LIN {X 0,Y 109.952,Z 432.134,A -85,B 0,C 180,E1 -30818.427,E2 -30818.427} C_VEL
LIN {X 0,Y 110.137,Z 438.588,A -85,B 0,C 180,E1 -30824.579,E2 -30824.579} C_VEL
LIN {X 0,Y 111.737,Z 444.355,A -85,B 0,C 180,E1 -30831.025,E2 -30831.025} C_VEL
LIN {X 0,Y 115.537,Z 449.975,A -85,B 0,C 180,E1 -30838.383,E2 -30838.383} C_VEL
LIN {X 0,Y 120.475,Z 454.059,A -85,B 0,C 180,E1 -30844.487,E2 -30844.487} C_VEL
LIN {X 0,Y 127.737,Z 457.673,A -85,B 0,C 180,E1 -30850.724,E2 -30850.724} C_VEL
LIN {X 0,Y 137.278,Z 460.508,A -85,B 0,C 180,E1 -30856.577,E2 -30856.577} C_VEL
LIN {X 0,Y 149.17,Z 462.456,A -85,B 0,C 180,E1 -30861.875,E2 -30861.875} C_VEL
LIN {X 0,Y 161.996,Z 463.408,A -85,B 0,C 180,E1 -30866.197,E2 -30866.197} C_VEL
LIN {X 0,Y 176.213,Z 463.483,A -85,B 0,C 180,E1 -30870,E2 -30870} C_VEL
LIN {X 0,Y 161.996,Z 463.408,A -85,B 0,C 180,E1 -30873.803,E2 -30873.803} C_VEL
LIN {X 0,Y 156.475,Z 463.174,A -85,B 0,C 180,E1 -30875.531,E2 -30875.531} C_VEL
LIN {X 0,Y 151.713,Z 462.95,A -85,B 0,C 180,E1 -30876.832,E2 -30876.832} C_VEL
LIN {X 0,Y 136.071,Z 462.302,A -85,B 0,C 180,E1 -30880.248,E2 -30880.248} C_VEL
LIN {X 0,Y 131.493,Z 461.883,A -85,B 0,C 180,E1 -30881.828,E2 -30881.828} C_VEL
LIN {X 0,Y 130.179,Z 461.635,A -85,B 0,C 180,E1 -30882.462,E2 -30882.462} C_VEL
LIN {X 0,Y 123.589,Z 460.079,A -85,B 0,C 180,E1 -30886.519,E2 -30886.519} C_VEL
LIN {X 0,Y 114.993,Z 456.749,A -85,B 0,C 180,E1 -30893.55,E2 -30893.55} C_VEL
LIN {X 0,Y 108.187,Z 451.587,A -85,B 0,C 180,E1 -30902.386,E2 -30902.386} C_VEL
LIN {X 0,Y 104.991,Z 446.653,A -85,B 0,C 180,E1 -30909.668,E2 -30909.668} C_VEL
LIN {X 0,Y 103.684,Z 440.506,A -85,B 0,C 180,E1 -30917.329,E2 -30917.329} C_VEL
LIN {X 0,Y 104.202,Z 433.989,A -85,B 0,C 180,E1 -30924.032,E2 -30924.032} C_VEL
LIN {X 0,Y 105.726,Z 427.305,A -85,B 0,C 180,E1 -30929.787,E2 -30929.787} C_VEL
LIN {X 0,Y 108.121,Z 419.38,A -85,B 0,C 180,E1 -30935.507,E2 -30935.507} C_VEL
LIN {X 0,Y 110.878,Z 411.533,A -85,B 0,C 180,E1 -30940.085,E2 -30940.085} C_VEL
LIN {X 0,Y 114.106,Z 402.226,A -85,B 0,C 180,E1 -30944.598,E2 -30944.598} C_VEL
LIN {X 0,Y 115.928,Z 396.712,A -85,B 0,C 180,E1 -30947.094,E2 -30947.094} C_VEL
LIN {X 0,Y 116.823,Z 392.5,A -85,B 0,C 180,E1 -30949.604,E2 -30949.604} C_VEL
LIN {X 0,Y 117.25,Z 390.258,A -85,B 0,C 180,E1 -30951.384,E2 -30951.384} C_VEL
LIN {X 0,Y 117.552,Z 388.558,A -85,B 0,C 180,E1 -30953.134,E2 -30953.134} C_VEL
LIN {X 0,Y 117.819,Z 386.305,A -85,B 0,C 180,E1 -30956.582,E2 -30956.582} C_VEL
LIN {X 0,Y 118.147,Z 384.922,A -85,B 0,C 180,E1 -30960.002,E2 -30960.002} C_VEL
LIN {X 0,Y 117.859,Z 385.79,A -85,B 0,C 180,E1 -30960.343,E2 -30960.343} C_VEL
LIN {X 0,Y 112.453,Z 398.556,A -85,B 0,C 180,E1 -30960.593,E2 -30960.593} C_VEL
LIN {X 0,Y 106.312,Z 409.458,A -85,B 0,C 180,E1 -30960.926,E2 -30960.926} C_VEL
LIN {X 0,Y 100.174,Z 418.396,A -85,B 0,C 180,E1 -30961.299,E2 -30961.299} C_VEL
LIN {X 0,Y 93.168,Z 426.918,A -85,B 0,C 180,E1 -30961.829,E2 -30961.829} C_VEL
LIN {X 0,Y 86.171,Z 434.13,A -85,B 0,C 180,E1 -30962.44,E2 -30962.44} C_VEL
LIN {X 0,Y 79.185,Z 440.325,A -85,B 0,C 180,E1 -30963.163,E2 -30963.163} C_VEL
LIN {X 0,Y 70.482,Z 446.858,A -85,B 0,C 180,E1 -30964.342,E2 -30964.342} C_VEL
LIN {X 0,Y 63.553,Z 451.36,A -85,B 0,C 180,E1 -30965.578,E2 -30965.578} C_VEL
LIN {X 0,Y 52.232,Z 457.31,A -85,B 0,C 180,E1 -30968.352,E2 -30968.352} C_VEL
LIN {X 0,Y 43.038,Z 461.18,A -85,B 0,C 180,E1 -30971.539,E2 -30971.539} C_VEL
LIN {X 0,Y 36.381,Z 463.552,A -85,B 0,C 180,E1 -30975.008,E2 -30975.008} C_VEL
LIN {X 0,Y 29.882,Z 465.355,A -85,B 0,C 180,E1 -30979.819,E2 -30979.819} C_VEL
LIN {X 0,Y 18.308,Z 467.822,A -85,B 0,C 180,E1 -30999.849,E2 -30999.849} C_VEL
LIN {X 0,Y 14.256,Z 468.423,A -85,B 0,C 180,E1 -31020.462,E2 -31020.462} C_VEL
LIN {X 0,Y 12.863,Z 468.588,A -85,B 0,C 180,E1 -31050,E2 -31050} C_VEL
LIN {X 0,Y 14.211,Z 468.422,A -85,B 0,C 180,E1 -31079.639,E2 -31079.639} C_VEL
LIN {X 0,Y 18.299,Z 467.822,A -85,B 0,C 180,E1 -31100.185,E2 -31100.185} C_VEL
LIN {X 0,Y 29.88,Z 465.354,A -85,B 0,C 180,E1 -31120.192,E2 -31120.192} C_VEL
LIN {X 0,Y 39.698,Z 462.4,A -85,B 0,C 180,E1 -31126.828,E2 -31126.828} C_VEL
LIN {X 0,Y 49.824,Z 458.409,A -85,B 0,C 180,E1 -31130.891,E2 -31130.891} C_VEL
LIN {X 0,Y 56.662,Z 455.192,A -85,B 0,C 180,E1 -31132.871,E2 -31132.871} C_VEL
LIN {X 0,Y 67.011,Z 449.168,A -85,B 0,C 180,E1 -31135.099,E2 -31135.099} C_VEL
LIN {X 0,Y 75.7,Z 443.075,A -85,B 0,C 180,E1 -31136.405,E2 -31136.405} C_VEL
LIN {X 0,Y 82.677,Z 437.38,A -85,B 0,C 180,E1 -31137.211,E2 -31137.211} C_VEL
LIN {X 0,Y 91.416,Z 428.834,A -85,B 0,C 180,E1 -31138.06,E2 -31138.06} C_VEL
LIN {X 0,Y 98.422,Z 420.664,A -85,B 0,C 180,E1 -31138.572,E2 -31138.572} C_VEL
LIN {X 0,Y 104.558,Z 412.16,A -85,B 0,C 180,E1 -31138.954,E2 -31138.954} C_VEL
LIN {X 0,Y 109.821,Z 403.451,A -85,B 0,C 180,E1 -31139.25,E2 -31139.25} C_VEL
LIN {X 0,Y 114.577,Z 393.86,A -85,B 0,C 180,E1 -31139.51,E2 -31139.51} C_VEL
LIN {X 0,Y 117.86,Z 385.789,A -85,B 0,C 180,E1 -31139.657,E2 -31139.657} C_VEL
LIN {X 0,Y 118.148,Z 384.921,A -85,B 0,C 180,E1 -31139.998,E2 -31139.998} C_VEL
LIN {X 0,Y 117.764,Z 386.797,A -85,B 0,C 180,E1 -31144.354,E2 -31144.354} C_VEL
LIN {X 0,Y 117.379,Z 389.446,A -85,B 0,C 180,E1 -31147.772,E2 -31147.772} C_VEL
LIN {X 0,Y 116.822,Z 392.502,A -85,B 0,C 180,E1 -31150.396,E2 -31150.396} C_VEL
LIN {X 0,Y 115.913,Z 396.746,A -85,B 0,C 180,E1 -31152.908,E2 -31152.908} C_VEL
LIN {X 0,Y 111.99,Z 408.401,A -85,B 0,C 180,E1 -31158.285,E2 -31158.285} C_VEL
LIN {X 0,Y 109.125,Z 416.544,A -85,B 0,C 180,E1 -31162.73,E2 -31162.73} C_VEL
LIN {X 0,Y 106.783,Z 423.698,A -85,B 0,C 180,E1 -31167.431,E2 -31167.431} C_VEL
LIN {X 0,Y 104.743,Z 431.236,A -85,B 0,C 180,E1 -31173.42,E2 -31173.42} C_VEL
LIN {X 0,Y 103.743,Z 438.536,A -85,B 0,C 180,E1 -31180.523,E2 -31180.523} C_VEL
LIN {X 0,Y 104.357,Z 444.73,A -85,B 0,C 180,E1 -31187.796,E2 -31187.796} C_VEL
LIN {X 0,Y 106.952,Z 450.021,A -85,B 0,C 180,E1 -31195.218,E2 -31195.218} C_VEL
LIN {X 0,Y 111.237,Z 454.336,A -85,B 0,C 180,E1 -31202.189,E2 -31202.189} C_VEL
LIN {X 0,Y 117.725,Z 457.962,A -85,B 0,C 180,E1 -31209.011,E2 -31209.011} C_VEL
LIN {X 0,Y 124.29,Z 460.275,A -85,B 0,C 180,E1 -31213.994,E2 -31213.994} C_VEL
LIN {X 0,Y 135.51,Z 462.499,A -85,B 0,C 180,E1 -31220.188,E2 -31220.188} C_VEL
LIN {X 0,Y 148.1,Z 463.65,A -85,B 0,C 180,E1 -31225.215,E2 -31225.215} C_VEL
LIN {X 0,Y 164.307,Z 463.8,A -85,B 0,C 180,E1 -31230,E2 -31230} C_VEL
LIN {X 0,Y 148.1,Z 463.65,A -85,B 0,C 180,E1 -31234.785,E2 -31234.785} C_VEL
LIN {X 0,Y 135.507,Z 462.502,A -85,B 0,C 180,E1 -31239.804,E2 -31239.804} C_VEL
LIN {X 0,Y 130.179,Z 461.635,A -85,B 0,C 180,E1 -31242.462,E2 -31242.462} C_VEL
LIN {X 0,Y 126.047,Z 461.085,A -85,B 0,C 180,E1 -31244.343,E2 -31244.343} C_VEL
LIN {X 0,Y 112.381,Z 459.488,A -85,B 0,C 180,E1 -31249.817,E2 -31249.817} C_VEL
LIN {X 0,Y 108.767,Z 458.593,A -85,B 0,C 180,E1 -31252.181,E2 -31252.181} C_VEL
LIN {X 0,Y 107.836,Z 458.22,A -85,B 0,C 180,E1 -31253.074,E2 -31253.074} C_VEL
LIN {X 0,Y 102.163,Z 454.476,A -85,B 0,C 180,E1 -31260.749,E2 -31260.749} C_VEL
LIN {X 0,Y 98.358,Z 449.147,A -85,B 0,C 180,E1 -31270.022,E2 -31270.022} C_VEL
LIN {X 0,Y 97.462,Z 442.32,A -85,B 0,C 180,E1 -31279.537,E2 -31279.537} C_VEL
LIN {X 0,Y 98.883,Z 435.097,A -85,B 0,C 180,E1 -31287.472,E2 -31287.472} C_VEL
LIN {X 0,Y 101.522,Z 427.548,A -85,B 0,C 180,E1 -31294.149,E2 -31294.149} C_VEL
LIN {X 0,Y 104.836,Z 419.614,A -85,B 0,C 180,E1 -31299.806,E2 -31299.806} C_VEL
LIN {X 0,Y 108.204,Z 411.945,A -85,B 0,C 180,E1 -31304.222,E2 -31304.222} C_VEL
LIN {X 0,Y 111.814,Z 403.367,A -85,B 0,C 180,E1 -31308.338,E2 -31308.338} C_VEL
LIN {X 0,Y 113.229,Z 399.587,A -85,B 0,C 180,E1 -31310.254,E2 -31310.254} C_VEL
LIN {X 0,Y 114.354,Z 395.938,A -85,B 0,C 180,E1 -31312.942,E2 -31312.942} C_VEL
LIN {X 0,Y 114.723,Z 394.314,A -85,B 0,C 180,E1 -31314.73,E2 -31314.73} C_VEL
LIN {X 0,Y 115.014,Z 393.125,A -85,B 0,C 180,E1 -31316.499,E2 -31316.499} C_VEL
LIN {X 0,Y 114.341,Z 394.573,A -85,B 0,C 180,E1 -31316.93,E2 -31316.93} C_VEL
LIN {X 0,Y 108.194,Z 406.499,A -85,B 0,C 180,E1 -31317.094,E2 -31317.094} C_VEL
LIN {X 0,Y 101.148,Z 417.069,A -85,B 0,C 180,E1 -31317.196,E2 -31317.196} C_VEL
LIN {X 0,Y 94.977,Z 424.806,A -85,B 0,C 180,E1 -31317.373,E2 -31317.373} C_VEL
LIN {X 0,Y 86.161,Z 433.937,A -85,B 0,C 180,E1 -31317.715,E2 -31317.715} C_VEL
LIN {X 0,Y 79.113,Z 440.132,A -85,B 0,C 180,E1 -31318.007,E2 -31318.007} C_VEL
LIN {X 0,Y 70.302,Z 446.665,A -85,B 0,C 180,E1 -31318.545,E2 -31318.545} C_VEL
LIN {X 0,Y 63.259,Z 451.166,A -85,B 0,C 180,E1 -31319.122,E2 -31319.122} C_VEL
LIN {X 0,Y 53.191,Z 456.446,A -85,B 0,C 180,E1 -31320.252,E2 -31320.252} C_VEL
LIN {X 0,Y 42.194,Z 460.986,A -85,B 0,C 180,E1 -31322.015,E2 -31322.015} C_VEL
LIN {X 0,Y 35.215,Z 463.358,A -85,B 0,C 180,E1 -31323.75,E2 -31323.75} C_VEL
LIN {X 0,Y 28.272,Z 465.161,A -85,B 0,C 180,E1 -31326.108,E2 -31326.108} C_VEL
LIN {X 0,Y 14.79,Z 467.629,A -85,B 0,C 180,E1 -31338.131,E2 -31338.131} C_VEL
LIN {X 0,Y 8.798,Z 468.23,A -85,B 0,C 180,E1 -31356.98,E2 -31356.98} C_VEL
LIN {X 0,Y 5.75,Z 468.395,A -85,B 0,C 180,E1 -31410,E2 -31410} C_VEL
LIN {X 0,Y 8.773,Z 468.229,A -85,B 0,C 180,E1 -31463.237,E2 -31463.237} C_VEL
LIN {X 0,Y 14.786,Z 467.628,A -85,B 0,C 180,E1 -31481.916,E2 -31481.916} C_VEL
LIN {X 0,Y 28.272,Z 465.161,A -85,B 0,C 180,E1 -31493.903,E2 -31493.903} C_VEL
LIN {X 0,Y 38.701,Z 462.206,A -85,B 0,C 180,E1 -31497.178,E2 -31497.178} C_VEL
LIN {X 0,Y 49.201,Z 458.215,A -85,B 0,C 180,E1 -31499.134,E2 -31499.134} C_VEL
LIN {X 0,Y 56.224,Z 454.998,A -85,B 0,C 180,E1 -31500.109,E2 -31500.109} C_VEL
LIN {X 0,Y 66.78,Z 448.975,A -85,B 0,C 180,E1 -31501.195,E2 -31501.195} C_VEL
LIN {X 0,Y 75.588,Z 442.882,A -85,B 0,C 180,E1 -31501.805,E2 -31501.805} C_VEL
LIN {X 0,Y 82.636,Z 437.188,A -85,B 0,C 180,E1 -31502.136,E2 -31502.136} C_VEL
LIN {X 0,Y 91.451,Z 428.641,A -85,B 0,C 180,E1 -31502.512,E2 -31502.512} C_VEL
LIN {X 0,Y 98.501,Z 420.471,A -85,B 0,C 180,E1 -31502.707,E2 -31502.707} C_VEL
LIN {X 0,Y 104.67,Z 411.967,A -85,B 0,C 180,E1 -31502.846,E2 -31502.846} C_VEL
LIN {X 0,Y 109.958,Z 403.259,A -85,B 0,C 180,E1 -31502.954,E2 -31502.954} C_VEL
LIN {X 0,Y 114.162,Z 394.978,A -85,B 0,C 180,E1 -31503.048,E2 -31503.048} C_VEL
LIN {X 0,Y 115.013,Z 393.127,A -85,B 0,C 180,E1 -31503.501,E2 -31503.501} C_VEL
LIN {X 0,Y 114.72,Z 394.322,A -85,B 0,C 180,E1 -31505.271,E2 -31505.271} C_VEL
LIN {X 0,Y 114.113,Z 396.913,A -85,B 0,C 180,E1 -31507.879,E2 -31507.879} C_VEL
LIN {X 0,Y 113.211,Z 399.616,A -85,B 0,C 180,E1 -31509.742,E2 -31509.742} C_VEL
LIN {X 0,Y 111.451,Z 404.34,A -85,B 0,C 180,E1 -31512.115,E2 -31512.115} C_VEL
LIN {X 0,Y 106.913,Z 415.068,A -85,B 0,C 180,E1 -31517.439,E2 -31517.439} C_VEL
LIN {X 0,Y 102.995,Z 423.979,A -85,B 0,C 180,E1 -31523.098,E2 -31523.098} C_VEL
LIN {X 0,Y 99.632,Z 432.65,A -85,B 0,C 180,E1 -31530.194,E2 -31530.194} C_VEL
LIN {X 0,Y 97.958,Z 438.802,A -85,B 0,C 180,E1 -31536.404,E2 -31536.404} C_VEL
LIN {X 0,Y 97.46,Z 444.88,A -85,B 0,C 180,E1 -31543.853,E2 -31543.853} C_VEL
LIN {X 0,Y 98.802,Z 450.027,A -85,B 0,C 180,E1 -31551.482,E2 -31551.482} C_VEL
LIN {X 0,Y 102.145,Z 454.481,A -85,B 0,C 180,E1 -31559.251,E2 -31559.251} C_VEL
LIN {X 0,Y 107.92,Z 458.249,A -85,B 0,C 180,E1 -31567,E2 -31567} C_VEL
LIN {X 0,Y 113.251,Z 460.373,A -85,B 0,C 180,E1 -31571.924,E2 -31571.924} C_VEL
LIN {X 0,Y 122.132,Z 462.491,A -85,B 0,C 180,E1 -31578.019,E2 -31578.019} C_VEL
LIN {X 0,Y 134.521,Z 463.877,A -85,B 0,C 180,E1 -31584.002,E2 -31584.002} C_VEL
LIN {X 0,Y 147.626,Z 464.245,A -85,B 0,C 180,E1 -31588.622,E2 -31588.622} C_VEL
LIN {X 0,Y 152.404,Z 464.117,A -85,B 0,C 180,E1 -31590,E2 -31590} C_VEL
LIN {X 0,Y 140.832,Z 464.131,A -85,B 0,C 180,E1 -31593.586,E2 -31593.586} C_VEL
LIN {X 0,Y 128.02,Z 463.258,A -85,B 0,C 180,E1 -31598.838,E2 -31598.838} C_VEL
LIN {X 0,Y 119.447,Z 461.928,A -85,B 0,C 180,E1 -31603.612,E2 -31603.612} C_VEL
LIN {X 0,Y 111.726,Z 459.855,A -85,B 0,C 180,E1 -31609.349,E2 -31609.349} C_VEL
LIN {X 0,Y 107.836,Z 458.22,A -85,B 0,C 180,E1 -31613.074,E2 -31613.074} C_VEL
LIN {X 0,Y 104.866,Z 457.195,A -85,B 0,C 180,E1 -31615.774,E2 -31615.774} C_VEL
LIN {X 0,Y 94.718,Z 454.51,A -85,B 0,C 180,E1 -31624.073,E2 -31624.073} C_VEL
LIN {X 0,Y 92.527,Z 453.084,A -85,B 0,C 180,E1 -31627.303,E2 -31627.303} C_VEL
LIN {X 0,Y 92.109,Z 452.483,A -85,B 0,C 180,E1 -31628.434,E2 -31628.434} C_VEL
LIN {X 0,Y 91.027,Z 448.147,A -85,B 0,C 180,E1 -31635.987,E2 -31635.987} C_VEL
LIN {X 0,Y 91.944,Z 441.68,A -85,B 0,C 180,E1 -31645.026,E2 -31645.026} C_VEL
LIN {X 0,Y 94.688,Z 434.482,A -85,B 0,C 180,E1 -31652.958,E2 -31652.958} C_VEL
LIN {X 0,Y 98.08,Z 427.57,A -85,B 0,C 180,E1 -31659.008,E2 -31659.008} C_VEL
LIN {X 0,Y 102.195,Z 419.847,A -85,B 0,C 180,E1 -31664.319,E2 -31664.319} C_VEL
LIN {X 0,Y 106.656,Z 411.289,A -85,B 0,C 180,E1 -31669.057,E2 -31669.057} C_VEL
LIN {X 0,Y 109.831,Z 404.885,A -85,B 0,C 180,E1 -31672.135,E2 -31672.135} C_VEL
LIN {X 0,Y 110.22,Z 403.943,A -85,B 0,C 180,E1 -31672.675,E2 -31672.675} C_VEL
LIN {X 0,Y 109.148,Z 405.657,A -85,B 0,C 180,E1 -31673.363,E2 -31673.363} C_VEL
LIN {X 0,Y 101.742,Z 416.876,A -85,B 0,C 180,E1 -31673.202,E2 -31673.202} C_VEL
LIN {X 0,Y 95.565,Z 424.614,A -85,B 0,C 180,E1 -31673.121,E2 -31673.121} C_VEL
LIN {X 0,Y 86.738,Z 433.743,A -85,B 0,C 180,E1 -31673.006,E2 -31673.006} C_VEL
LIN {X 0,Y 79.68,Z 439.938,A -85,B 0,C 180,E1 -31672.876,E2 -31672.876} C_VEL
LIN {X 0,Y 70.844,Z 446.471,A -85,B 0,C 180,E1 -31672.763,E2 -31672.763} C_VEL
LIN {X 0,Y 63.769,Z 450.972,A -85,B 0,C 180,E1 -31672.696,E2 -31672.696} C_VEL
LIN {X 0,Y 52.644,Z 456.689,A -85,B 0,C 180,E1 -31672.586,E2 -31672.586} C_VEL
LIN {X 0,Y 42.543,Z 460.793,A -85,B 0,C 180,E1 -31672.387,E2 -31672.387} C_VEL
LIN {X 0,Y 35.468,Z 463.165,A -85,B 0,C 180,E1 -31672.197,E2 -31672.197} C_VEL
LIN {X 0,Y 28.411,Z 464.968,A -85,B 0,C 180,E1 -31671.683,E2 -31671.683} C_VEL
LIN {X 0,Y 14.284,Z 467.435,A -85,B 0,C 180,E1 -31669.75,E2 -31669.75} C_VEL
LIN {X 0,Y 7.265,Z 468.037,A -85,B 0,C 180,E1 -31665.329,E2 -31665.329} C_VEL
LIN {X 0,Y 1.35,Z 468.202,A -85,B 0,C 180,E1 -31590,E2 -31590} C_VEL
LIN {X 0,Y 7.274,Z 468.036,A -85,B 0,C 180,E1 -31514.948,E2 -31514.948} C_VEL
LIN {X 0,Y 14.286,Z 467.434,A -85,B 0,C 180,E1 -31510.299,E2 -31510.299} C_VEL
LIN {X 0,Y 28.411,Z 464.968,A -85,B 0,C 180,E1 -31508.326,E2 -31508.326} C_VEL
LIN {X 0,Y 39.008,Z 462.012,A -85,B 0,C 180,E1 -31507.727,E2 -31507.727} C_VEL
LIN {X 0,Y 49.609,Z 458.021,A -85,B 0,C 180,E1 -31507.405,E2 -31507.405} C_VEL
LIN {X 0,Y 56.686,Z 454.805,A -85,B 0,C 180,E1 -31507.326,E2 -31507.326} C_VEL
LIN {X 0,Y 67.307,Z 448.782,A -85,B 0,C 180,E1 -31507.273,E2 -31507.273} C_VEL
LIN {X 0,Y 76.145,Z 442.689,A -85,B 0,C 180,E1 -31507.166,E2 -31507.166} C_VEL
LIN {X 0,Y 83.204,Z 436.995,A -85,B 0,C 180,E1 -31507.031,E2 -31507.031} C_VEL
LIN {X 0,Y 92.036,Z 428.448,A -85,B 0,C 180,E1 -31506.932,E2 -31506.932} C_VEL
LIN {X 0,Y 99.092,Z 420.278,A -85,B 0,C 180,E1 -31506.818,E2 -31506.818} C_VEL
LIN {X 0,Y 105.262,Z 411.774,A -85,B 0,C 180,E1 -31506.712,E2 -31506.712} C_VEL
LIN {X 0,Y 109.135,Z 405.681,A -85,B 0,C 180,E1 -31506.638,E2 -31506.638} C_VEL
LIN {X 0,Y 110.199,Z 403.982,A -85,B 0,C 180,E1 -31507.326,E2 -31507.326} C_VEL
LIN {X 0,Y 108.098,Z 408.486,A -85,B 0,C 180,E1 -31509.608,E2 -31509.608} C_VEL
LIN {X 0,Y 103.808,Z 416.836,A -85,B 0,C 180,E1 -31513.852,E2 -31513.852} C_VEL
LIN {X 0,Y 99.108,Z 425.627,A -85,B 0,C 180,E1 -31519.53,E2 -31519.53} C_VEL
LIN {X 0,Y 95.44,Z 432.915,A -85,B 0,C 180,E1 -31525.575,E2 -31525.575} C_VEL
LIN {X 0,Y 92.739,Z 439.22,A -85,B 0,C 180,E1 -31532.035,E2 -31532.035} C_VEL
LIN {X 0,Y 91.166,Z 445.137,A -85,B 0,C 180,E1 -31539.565,E2 -31539.565} C_VEL
LIN {X 0,Y 91.301,Z 450.221,A -85,B 0,C 180,E1 -31547.509,E2 -31547.509} C_VEL
LIN {X 0,Y 93.529,Z 454.579,A -85,B 0,C 180,E1 -31555.743,E2 -31555.743} C_VEL
LIN {X 0,Y 98.452,Z 458.531,A -85,B 0,C 180,E1 -31564.64,E2 -31564.64} C_VEL
LIN {X 0,Y 104.083,Z 460.927,A -85,B 0,C 180,E1 -31570.959,E2 -31570.959} C_VEL
LIN {X 0,Y 114.583,Z 463.243,A -85,B 0,C 180,E1 -31578.912,E2 -31578.912} C_VEL
LIN {X 0,Y 123.076,Z 464.184,A -85,B 0,C 180,E1 -31583.442,E2 -31583.442} C_VEL
LIN {X 0,Y 133.634,Z 464.587,A -85,B 0,C 180,E1 -31587.718,E2 -31587.718} C_VEL
LIN {X 0,Y 140.49,Z 464.434,A -85,B 0,C 180,E1 -31590,E2 -31590} C_VEL
LIN {X 0,Y 131.483,Z 464.526,A -85,B 0,C 180,E1 -31593.064,E2 -31593.064} C_VEL
LIN {X 0,Y 120.584,Z 464.003,A -85,B 0,C 180,E1 -31597.787,E2 -31597.787} C_VEL
LIN {X 0,Y 108.959,Z 462.222,A -85,B 0,C 180,E1 -31604.952,E2 -31604.952} C_VEL
LIN {X 0,Y 101.593,Z 460.006,A -85,B 0,C 180,E1 -31611.561,E2 -31611.561} C_VEL
LIN {X 0,Y 94.865,Z 455.993,A -85,B 0,C 180,E1 -31621.238,E2 -31621.238} C_VEL
LIN {X 0,Y 92.109,Z 452.483,A -85,B 0,C 180,E1 -31628.434,E2 -31628.434} C_VEL
LIN {X 0,Y 90.747,Z 450.813,A -85,B 0,C 180,E1 -31631.881,E2 -31631.881} C_VEL
LIN {X 0,Y 86.069,Z 446.561,A -85,B 0,C 180,E1 -31642.687,E2 -31642.687} C_VEL
LIN {X 0,Y 85.932,Z 444.588,A -85,B 0,C 180,E1 -31646.376,E2 -31646.376} C_VEL
LIN {X 0,Y 86.196,Z 443.807,A -85,B 0,C 180,E1 -31647.559,E2 -31647.559} C_VEL
LIN {X 0,Y 89.395,Z 437.538,A -85,B 0,C 180,E1 -31655.199,E2 -31655.199} C_VEL
LIN {X 0,Y 94.292,Z 429.466,A -85,B 0,C 180,E1 -31662.657,E2 -31662.657} C_VEL
LIN {X 0,Y 99.457,Z 421.341,A -85,B 0,C 180,E1 -31668.293,E2 -31668.293} C_VEL
LIN {X 0,Y 100.189,Z 420.084,A -85,B 0,C 180,E1 -31669.131,E2 -31669.131} C_VEL
LIN {X 0,Y 93.163,Z 428.255,A -85,B 0,C 180,E1 -31668.722,E2 -31668.722} C_VEL
LIN {X 0,Y 84.379,Z 436.801,A -85,B 0,C 180,E1 -31668.143,E2 -31668.143} C_VEL
LIN {X 0,Y 73.842,Z 445.123,A -85,B 0,C 180,E1 -31667.304,E2 -31667.304} C_VEL
LIN {X 0,Y 65.059,Z 450.779,A -85,B 0,C 180,E1 -31666.464,E2 -31666.464} C_VEL
LIN {X 0,Y 55.042,Z 456.046,A -85,B 0,C 180,E1 -31665.209,E2 -31665.209} C_VEL
LIN {X 0,Y 47.52,Z 459.36,A -85,B 0,C 180,E1 -31664.01,E2 -31664.01} C_VEL
LIN {X 0,Y 37.118,Z 462.971,A -85,B 0,C 180,E1 -31661.211,E2 -31661.211} C_VEL
LIN {X 0,Y 23.545,Z 466.17,A -85,B 0,C 180,E1 -31653.571,E2 -31653.571} C_VEL
LIN {X 0,Y 17.066,Z 467.241,A -85,B 0,C 180,E1 -31645.448,E2 -31645.448} C_VEL
LIN {X 0,Y 11.39,Z 467.843,A -85,B 0,C 180,E1 -31628.098,E2 -31628.098} C_VEL
LIN {X 0,Y 8.44,Z 468.01,A -85,B 0,C 180,E1 -31590,E2 -31590} C_VEL
LIN {X 0,Y 11.414,Z 467.843,A -85,B 0,C 180,E1 -31551.995,E2 -31551.995} C_VEL
LIN {X 0,Y 17.073,Z 467.241,A -85,B 0,C 180,E1 -31534.583,E2 -31534.583} C_VEL
LIN {X 0,Y 30.271,Z 464.775,A -85,B 0,C 180,E1 -31521.769,E2 -31521.769} C_VEL
LIN {X 0,Y 40.59,Z 461.818,A -85,B 0,C 180,E1 -31517.77,E2 -31517.77} C_VEL
LIN {X 0,Y 51.028,Z 457.827,A -85,B 0,C 180,E1 -31515.4,E2 -31515.4} C_VEL
LIN {X 0,Y 61.544,Z 452.695,A -85,B 0,C 180,E1 -31513.916,E2 -31513.916} C_VEL
LIN {X 0,Y 70.329,Z 447.433,A -85,B 0,C 180,E1 -31513.014,E2 -31513.014} C_VEL
LIN {X 0,Y 79.112,Z 441.12,A -85,B 0,C 180,E1 -31512.262,E2 -31512.262} C_VEL
LIN {X 0,Y 86.133,Z 435.175,A -85,B 0,C 180,E1 -31511.727,E2 -31511.727} C_VEL
LIN {X 0,Y 93.162,Z 428.255,A -85,B 0,C 180,E1 -31511.275,E2 -31511.275} C_VEL
LIN {X 0,Y 100.187,Z 420.084,A -85,B 0,C 180,E1 -31510.864,E2 -31510.864} C_VEL
LIN {X 0,Y 95.171,Z 428.026,A -85,B 0,C 180,E1 -31516.261,E2 -31516.261} C_VEL
LIN {X 0,Y 90.494,Z 435.565,A -85,B 0,C 180,E1 -31522.847,E2 -31522.847} C_VEL
LIN {X 0,Y 86.415,Z 443.315,A -85,B 0,C 180,E1 -31531.743,E2 -31531.743} C_VEL
LIN {X 0,Y 84.543,Z 449.726,A -85,B 0,C 180,E1 -31541.681,E2 -31541.681} C_VEL
LIN {X 0,Y 85.378,Z 454.613,A -85,B 0,C 180,E1 -31551.436,E2 -31551.436} C_VEL
LIN {X 0,Y 89.356,Z 458.807,A -85,B 0,C 180,E1 -31561.842,E2 -31561.842} C_VEL
LIN {X 0,Y 93.403,Z 460.947,A -85,B 0,C 180,E1 -31567.9,E2 -31567.9} C_VEL
LIN {X 0,Y 101.462,Z 463.165,A -85,B 0,C 180,E1 -31575.859,E2 -31575.859} C_VEL
LIN {X 0,Y 113.189,Z 464.541,A -85,B 0,C 180,E1 -31583.421,E2 -31583.421} C_VEL
LIN {X 0,Y 126.513,Z 464.807,A -85,B 0,C 180,E1 -31589.181,E2 -31589.181} C_VEL
LIN {X 0,Y 128.831,Z 464.745,A -85,B 0,C 180,E1 -31590,E2 -31590} C_VEL
LIN {X 0,Y 119.694,Z 464.822,A -85,B 0,C 180,E1 -31593.489,E2 -31593.489} C_VEL
LIN {X 0,Y 107.081,Z 463.973,A -85,B 0,C 180,E1 -31600.118,E2 -31600.118} C_VEL
LIN {X 0,Y 98.651,Z 462.513,A -85,B 0,C 180,E1 -31606.557,E2 -31606.557} C_VEL
LIN {X 0,Y 92.14,Z 460.392,A -85,B 0,C 180,E1 -31613.758,E2 -31613.758} C_VEL
LIN {X 0,Y 86.432,Z 456.265,A -85,B 0,C 180,E1 -31624.693,E2 -31624.693} C_VEL
LIN {X 0,Y 84.475,Z 451.478,A -85,B 0,C 180,E1 -31634.999,E2 -31634.999} C_VEL
LIN {X 0,Y 85.077,Z 446.713,A -85,B 0,C 180,E1 -31643.25,E2 -31643.25} C_VEL
LIN {X 0,Y 86.196,Z 443.807,A -85,B 0,C 180,E1 -31647.559,E2 -31647.559} C_VEL
LIN {X 0,Y 86.44,Z 442.413,A -85,B 0,C 180,E1 -31650.046,E2 -31650.046} C_VEL
LIN {X 0,Y 85.502,Z 439.043,A -85,B 0,C 180,E1 -31658.747,E2 -31658.747} C_VEL
LIN {X 0,Y 86.371,Z 437.319,A -85,B 0,C 180,E1 -31661.062,E2 -31661.062} C_VEL
LIN {X 0,Y 88.035,Z 434.965,A -85,B 0,C 180,E1 -31663.332,E2 -31663.332} C_VEL
LIN {X 0,Y 87.865,Z 434.982,A -85,B 0,C 180,E1 -31663.706,E2 -31663.706} C_VEL
LIN {X 0,Y 80.927,Z 440.927,A -85,B 0,C 180,E1 -31662.801,E2 -31662.801} C_VEL
LIN {X 0,Y 72.272,Z 447.24,A -85,B 0,C 180,E1 -31661.464,E2 -31661.464} C_VEL
LIN {X 0,Y 63.64,Z 452.501,A -85,B 0,C 180,E1 -31659.832,E2 -31659.832} C_VEL
LIN {X 0,Y 53.37,Z 457.633,A -85,B 0,C 180,E1 -31657.189,E2 -31657.189} C_VEL
LIN {X 0,Y 43.302,Z 461.624,A -85,B 0,C 180,E1 -31653.208,E2 -31653.208} C_VEL
LIN {X 0,Y 33.561,Z 464.582,A -85,B 0,C 180,E1 -31646.891,E2 -31646.891} C_VEL
LIN {X 0,Y 21.911,Z 467.047,A -85,B 0,C 180,E1 -31629.904,E2 -31629.904} C_VEL
LIN {X 0,Y 17.547,Z 467.65,A -85,B 0,C 180,E1 -31613.611,E2 -31613.611} C_VEL
LIN {X 0,Y 15.549,Z 467.817,A -85,B 0,C 180,E1 -31590,E2 -31590} C_VEL
LIN {X 0,Y 17.57,Z 467.65,A -85,B 0,C 180,E1 -31566.422,E2 -31566.422} C_VEL
LIN {X 0,Y 21.919,Z 467.047,A -85,B 0,C 180,E1 -31550.113,E2 -31550.113} C_VEL
LIN {X 0,Y 33.563,Z 464.582,A -85,B 0,C 180,E1 -31533.115,E2 -31533.115} C_VEL
LIN {X 0,Y 43.304,Z 461.624,A -85,B 0,C 180,E1 -31526.796,E2 -31526.796} C_VEL
LIN {X 0,Y 53.369,Z 457.633,A -85,B 0,C 180,E1 -31522.809,E2 -31522.809} C_VEL
LIN {X 0,Y 63.641,Z 452.501,A -85,B 0,C 180,E1 -31520.17,E2 -31520.17} C_VEL
LIN {X 0,Y 72.272,Z 447.24,A -85,B 0,C 180,E1 -31518.536,E2 -31518.536} C_VEL
LIN {X 0,Y 80.921,Z 440.927,A -85,B 0,C 180,E1 -31517.188,E2 -31517.188} C_VEL
LIN {X 0,Y 87.853,Z 434.983,A -85,B 0,C 180,E1 -31516.268,E2 -31516.268} C_VEL
LIN {X 0,Y 88.03,Z 434.966,A -85,B 0,C 180,E1 -31516.659,E2 -31516.659} C_VEL
LIN {X 0,Y 82.482,Z 442.715,A -85,B 0,C 180,E1 -31525.213,E2 -31525.213} C_VEL
LIN {X 0,Y 78.589,Z 449.926,A -85,B 0,C 180,E1 -31536.405,E2 -31536.405} C_VEL
LIN {X 0,Y 77.913,Z 454.583,A -85,B 0,C 180,E1 -31546.184,E2 -31546.184} C_VEL
LIN {X 0,Y 80.624,Z 459.081,A -85,B 0,C 180,E1 -31558.465,E2 -31558.465} C_VEL
LIN {X 0,Y 84.527,Z 461.44,A -85,B 0,C 180,E1 -31566.142,E2 -31566.142} C_VEL
LIN {X 0,Y 88.803,Z 462.864,A -85,B 0,C 180,E1 -31571.741,E2 -31571.741} C_VEL
LIN {X 0,Y 101.121,Z 464.785,A -85,B 0,C 180,E1 -31582.01,E2 -31582.01} C_VEL
LIN {X 0,Y 112.511,Z 465.186,A -85,B 0,C 180,E1 -31588.022,E2 -31588.022} C_VEL
LIN {X 0,Y 117.267,Z 465.056,A -85,B 0,C 180,E1 -31590,E2 -31590} C_VEL
LIN {X 0,Y 105.857,Z 465.007,A -85,B 0,C 180,E1 -31595.234,E2 -31595.234} C_VEL
LIN {X 0,Y 99.612,Z 464.684,A -85,B 0,C 180,E1 -31598.993,E2 -31598.993} C_VEL
LIN {X 0,Y 88.566,Z 462.8,A -85,B 0,C 180,E1 -31608.506,E2 -31608.506} C_VEL
LIN {X 0,Y 84.02,Z 461.224,A -85,B 0,C 180,E1 -31614.723,E2 -31614.723} C_VEL
LIN {X 0,Y 78.947,Z 457.333,A -85,B 0,C 180,E1 -31626.76,E2 -31626.76} C_VEL
LIN {X 0,Y 77.855,Z 453.539,A -85,B 0,C 180,E1 -31636.233,E2 -31636.233} C_VEL
LIN {X 0,Y 79.399,Z 448.009,A -85,B 0,C 180,E1 -31646.882,E2 -31646.882} C_VEL
LIN {X 0,Y 83.132,Z 441.707,A -85,B 0,C 180,E1 -31656.033,E2 -31656.033} C_VEL
LIN {X 0,Y 86.371,Z 437.319,A -85,B 0,C 180,E1 -31661.062,E2 -31661.062} C_VEL
LIN {X 0,Y 85.41,Z 438.095,A -85,B 0,C 180,E1 -31661.09,E2 -31661.09} C_VEL
LIN {X 0,Y 81.573,Z 441.77,A -85,B 0,C 180,E1 -31658.88,E2 -31658.88} C_VEL
LIN {X 0,Y 77.828,Z 445.591,A -85,B 0,C 180,E1 -31655.18,E2 -31655.18} C_VEL
LIN {X 0,Y 75.269,Z 448.303,A -85,B 0,C 180,E1 -31651.87,E2 -31651.87} C_VEL
LIN {X 0,Y 72.487,Z 451.757,A -85,B 0,C 180,E1 -31646.161,E2 -31646.161} C_VEL
LIN {X 0,Y 71.958,Z 452.745,A -85,B 0,C 180,E1 -31644.076,E2 -31644.076} C_VEL
LIN {X 0,Y 71.151,Z 456.799,A -85,B 0,C 180,E1 -31633.743,E2 -31633.743} C_VEL
LIN {X 0,Y 72.261,Z 459.353,A -85,B 0,C 180,E1 -31625.701,E2 -31625.701} C_VEL
LIN {X 0,Y 74.897,Z 461.5,A -85,B 0,C 180,E1 -31617.981,E2 -31617.981} C_VEL
LIN {X 0,Y 81.174,Z 463.741,A -85,B 0,C 180,E1 -31607.764,E2 -31607.764} C_VEL
LIN {X 0,Y 92.19,Z 465.166,A -85,B 0,C 180,E1 -31597.695,E2 -31597.695} C_VEL
LIN {X 0,Y 98.592,Z 465.473,A -85,B 0,C 180,E1 -31593.683,E2 -31593.683} C_VEL
LIN {X 0,Y 105.989,Z 465.362,A -85,B 0,C 180,E1 -31590,E2 -31590} C_VEL
LIN {X 0,Y 97.797,Z 465.439,A -85,B 0,C 180,E1 -31585.879,E2 -31585.879} C_VEL
LIN {X 0,Y 86.329,Z 464.603,A -85,B 0,C 180,E1 -31577.651,E2 -31577.651} C_VEL
LIN {X 0,Y 78.859,Z 463.079,A -85,B 0,C 180,E1 -31569.116,E2 -31569.116} C_VEL
LIN {X 0,Y 73.735,Z 460.696,A -85,B 0,C 180,E1 -31559.068,E2 -31559.068} C_VEL
LIN {X 0,Y 71.162,Z 456.799,A -85,B 0,C 180,E1 -31546.265,E2 -31546.265} C_VEL
LIN {X 0,Y 71.991,Z 452.703,A -85,B 0,C 180,E1 -31535.851,E2 -31535.851} C_VEL
LIN {X 0,Y 74.872,Z 448.093,A -85,B 0,C 180,E1 -31526.909,E2 -31526.909} C_VEL
LIN {X 0,Y 76.524,Z 445.892,A -85,B 0,C 180,E1 -31523.307,E2 -31523.307} C_VEL
LIN {X 0,Y 69.791,Z 450.391,A -85,B 0,C 180,E1 -31525.001,E2 -31525.001} C_VEL
LIN {X 0,Y 60.888,Z 455.367,A -85,B 0,C 180,E1 -31527.758,E2 -31527.758} C_VEL
LIN {X 0,Y 50.063,Z 460.214,A -85,B 0,C 180,E1 -31532.617,E2 -31532.617} C_VEL
LIN {X 0,Y 43.866,Z 462.583,A -85,B 0,C 180,E1 -31536.767,E2 -31536.767} C_VEL
LIN {X 0,Y 37.938,Z 464.388,A -85,B 0,C 180,E1 -31542.183,E2 -31542.183} C_VEL
LIN {X 0,Y 27.761,Z 466.854,A -85,B 0,C 180,E1 -31559.581,E2 -31559.581} C_VEL
LIN {X 0,Y 24.275,Z 467.456,A -85,B 0,C 180,E1 -31573.171,E2 -31573.171} C_VEL
LIN {X 0,Y 22.647,Z 467.624,A -85,B 0,C 180,E1 -31590,E2 -31590} C_VEL
LIN {X 0,Y 24.255,Z 467.457,A -85,B 0,C 180,E1 -31606.843,E2 -31606.843} C_VEL
LIN {X 0,Y 27.753,Z 466.854,A -85,B 0,C 180,E1 -31620.429,E2 -31620.429} C_VEL
LIN {X 0,Y 37.935,Z 464.388,A -85,B 0,C 180,E1 -31637.821,E2 -31637.821} C_VEL
LIN {X 0,Y 46.947,Z 461.431,A -85,B 0,C 180,E1 -31645.421,E2 -31645.421} C_VEL
LIN {X 0,Y 56.524,Z 457.439,A -85,B 0,C 180,E1 -31650.5,E2 -31650.5} C_VEL
LIN {X 0,Y 66.439,Z 452.307,A -85,B 0,C 180,E1 -31654.045,E2 -31654.045} C_VEL
LIN {X 0,Y 74.839,Z 447.046,A -85,B 0,C 180,E1 -31656.292,E2 -31656.292} C_VEL
LIN {X 0,Y 76.575,Z 445.888,A -85,B 0,C 180,E1 -31656.606,E2 -31656.606} C_VEL
LIN {X 0,Y 72.481,Z 451.702,A -85,B 0,C 180,E1 -31646.294,E2 -31646.294} C_VEL
LIN {X 0,Y 71.958,Z 452.745,A -85,B 0,C 180,E1 -31644.076,E2 -31644.076} C_VEL
LIN {X 0,Y 70.698,Z 454.879,A -85,B 0,C 180,E1 -31639.741,E2 -31639.741} C_VEL
LIN {X 0,Y 67.834,Z 458.333,A -85,B 0,C 180,E1 -31632.398,E2 -31632.398} C_VEL
LIN {X 0,Y 66.251,Z 461.115,A -85,B 0,C 180,E1 -31624.428,E2 -31624.428} C_VEL
LIN {X 0,Y 67.028,Z 462.248,A -85,B 0,C 180,E1 -31619.527,E2 -31619.527} C_VEL
LIN {X 0,Y 74.014,Z 464.529,A -85,B 0,C 180,E1 -31606.551,E2 -31606.551} C_VEL
LIN {X 0,Y 79.974,Z 465.366,A -85,B 0,C 180,E1 -31600.123,E2 -31600.123} C_VEL
LIN {X 0,Y 91.41,Z 465.759,A -85,B 0,C 180,E1 -31591.893,E2 -31591.893} C_VEL
LIN {X 0,Y 94.915,Z 465.662,A -85,B 0,C 180,E1 -31590,E2 -31590} C_VEL
LIN {X 0,Y 84.814,Z 465.631,A -85,B 0,C 180,E1 -31583.886,E2 -31583.886} C_VEL
LIN {X 0,Y 78.807,Z 465.287,A -85,B 0,C 180,E1 -31578.792,E2 -31578.792} C_VEL
LIN {X 0,Y 69.302,Z 463.308,A -85,B 0,C 180,E1 -31565.874,E2 -31565.874} C_VEL
LIN {X 0,Y 65.254,Z 460.777,A -85,B 0,C 180,E1 -31553.843,E2 -31553.843} C_VEL
LIN {X 0,Y 64.361,Z 458.555,A -85,B 0,C 180,E1 -31545.03,E2 -31545.03} C_VEL
LIN {X 0,Y 65.589,Z 454.96,A -85,B 0,C 180,E1 -31534.145,E2 -31534.145} C_VEL
LIN {X 0,Y 61.601,Z 456.625,A -85,B 0,C 180,E1 -31534.777,E2 -31534.777} C_VEL
LIN {X 0,Y 54.232,Z 460.02,A -85,B 0,C 180,E1 -31538.963,E2 -31538.963} C_VEL
LIN {X 0,Y 48.48,Z 462.389,A -85,B 0,C 180,E1 -31543.545,E2 -31543.545} C_VEL
LIN {X 0,Y 43.054,Z 464.194,A -85,B 0,C 180,E1 -31549.236,E2 -31549.236} C_VEL
LIN {X 0,Y 34.106,Z 466.66,A -85,B 0,C 180,E1 -31565.661,E2 -31565.661} C_VEL
LIN {X 0,Y 31.16,Z 467.263,A -85,B 0,C 180,E1 -31576.965,E2 -31576.965} C_VEL
LIN {X 0,Y 29.762,Z 467.431,A -85,B 0,C 180,E1 -31590,E2 -31590} C_VEL
LIN {X 0,Y 31.142,Z 467.263,A -85,B 0,C 180,E1 -31603.042,E2 -31603.042} C_VEL
LIN {X 0,Y 34.098,Z 466.66,A -85,B 0,C 180,E1 -31614.345,E2 -31614.345} C_VEL
LIN {X 0,Y 43.052,Z 464.194,A -85,B 0,C 180,E1 -31630.766,E2 -31630.766} C_VEL
LIN {X 0,Y 51.324,Z 461.237,A -85,B 0,C 180,E1 -31638.863,E2 -31638.863} C_VEL
LIN {X 0,Y 60.363,Z 457.245,A -85,B 0,C 180,E1 -31644.587,E2 -31644.587} C_VEL
LIN {X 0,Y 61.392,Z 456.736,A -85,B 0,C 180,E1 -31645.088,E2 -31645.088} C_VEL
LIN {X 0,Y 65.575,Z 454.966,A -85,B 0,C 180,E1 -31645.855,E2 -31645.855} C_VEL
LIN {X 0,Y 64.35,Z 458.554,A -85,B 0,C 180,E1 -31634.983,E2 -31634.983} C_VEL
LIN {X 0,Y 67.028,Z 462.248,A -85,B 0,C 180,E1 -31619.527,E2 -31619.527} C_VEL
LIN {X 0,Y 68.325,Z 463.31,A -85,B 0,C 180,E1 -31614.71,E2 -31614.71} C_VEL
LIN {X 0,Y 69.892,Z 464.809,A -85,B 0,C 180,E1 -31606.675,E2 -31606.675} C_VEL
LIN {X 0,Y 72.051,Z 465.651,A -85,B 0,C 180,E1 -31600.567,E2 -31600.567} C_VEL
LIN {X 0,Y 74.903,Z 465.946,A -85,B 0,C 180,E1 -31596.564,E2 -31596.564} C_VEL
LIN {X 0,Y 76.151,Z 466.015,A -85,B 0,C 180,E1 -31595.42,E2 -31595.42} C_VEL
LIN {X 0,Y 83.963,Z 465.96,A -85,B 0,C 180,E1 -31590,E2 -31590} C_VEL
LIN {X 0,Y 76.292,Z 466.025,A -85,B 0,C 180,E1 -31584.714,E2 -31584.714} C_VEL
LIN {X 0,Y 65.954,Z 465.137,A -85,B 0,C 180,E1 -31573.532,E2 -31573.532} C_VEL
LIN {X 0,Y 60.395,Z 463.628,A -85,B 0,C 180,E1 -31562.26,E2 -31562.26} C_VEL
LIN {X 0,Y 57.56,Z 460.827,A -85,B 0,C 180,E1 -31547.099,E2 -31547.099} C_VEL
LIN {X 0,Y 53.646,Z 462.195,A -85,B 0,C 180,E1 -31549.078,E2 -31549.078} C_VEL
LIN {X 0,Y 48.678,Z 464.001,A -85,B 0,C 180,E1 -31554.725,E2 -31554.725} C_VEL
LIN {X 0,Y 40.725,Z 466.466,A -85,B 0,C 180,E1 -31569.81,E2 -31569.81} C_VEL
LIN {X 0,Y 38.124,Z 467.07,A -85,B 0,C 180,E1 -31579.377,E2 -31579.377} C_VEL
LIN {X 0,Y 36.867,Z 467.238,A -85,B 0,C 180,E1 -31590,E2 -31590} C_VEL
LIN {X 0,Y 38.109,Z 467.07,A -85,B 0,C 180,E1 -31600.627,E2 -31600.627} C_VEL
LIN {X 0,Y 40.698,Z 466.467,A -85,B 0,C 180,E1 -31610.204,E2 -31610.204} C_VEL
LIN {X 0,Y 48.675,Z 464.001,A -85,B 0,C 180,E1 -31625.278,E2 -31625.278} C_VEL
LIN {X 0,Y 53.644,Z 462.196,A -85,B 0,C 180,E1 -31630.924,E2 -31630.924} C_VEL
LIN {X 0,Y 57.545,Z 460.835,A -85,B 0,C 180,E1 -31632.886,E2 -31632.886} C_VEL
LIN {X 0,Y 60.36,Z 463.63,A -85,B 0,C 180,E1 -31617.758,E2 -31617.758} C_VEL
LIN {X 0,Y 69.642,Z 465.652,A -85,B 0,C 180,E1 -31601.644,E2 -31601.644} C_VEL
LIN {X 0,Y 76.151,Z 466.015,A -85,B 0,C 180,E1 -31595.42,E2 -31595.42} C_VEL
LIN {X 0,Y 76.73,Z 466.125,A -85,B 0,C 180,E1 -31594.122,E2 -31594.122} C_VEL
LIN {X 0,Y 76.162,Z 466.18,A -85,B 0,C 180,E1 -31592.282,E2 -31592.282} C_VEL
LIN {X 0,Y 74.051,Z 466.272,A -85,B 0,C 180,E1 -31589.832,E2 -31589.832} C_VEL
LIN {X 0,Y 63.39,Z 466.175,A -85,B 0,C 180,E1 -31581.323,E2 -31581.323} C_VEL
LIN {X 0,Y 58.377,Z 465.81,A -85,B 0,C 180,E1 -31574.377,E2 -31574.377} C_VEL
LIN {X 0,Y 53.369,Z 464.675,A -85,B 0,C 180,E1 -31563.288,E2 -31563.288} C_VEL
LIN {X 0,Y 50.742,Z 465.202,A -85,B 0,C 180,E1 -31565.449,E2 -31565.449} C_VEL
LIN {X 0,Y 47.496,Z 466.272,A -85,B 0,C 180,E1 -31572.786,E2 -31572.786} C_VEL
LIN {X 0,Y 45.147,Z 466.876,A -85,B 0,C 180,E1 -31581.044,E2 -31581.044} C_VEL
LIN {X 0,Y 43.963,Z 467.046,A -85,B 0,C 180,E1 -31590,E2 -31590} C_VEL
LIN {X 0,Y 45.115,Z 466.877,A -85,B 0,C 180,E1 -31598.962,E2 -31598.962} C_VEL
LIN {X 0,Y 47.47,Z 466.273,A -85,B 0,C 180,E1 -31607.223,E2 -31607.223} C_VEL
LIN {X 0,Y 50.736,Z 465.202,A -85,B 0,C 180,E1 -31614.555,E2 -31614.555} C_VEL
LIN {X 0,Y 53.35,Z 464.681,A -85,B 0,C 180,E1 -31616.679,E2 -31616.679} C_VEL
LIN {X 0,Y 59.614,Z 465.931,A -85,B 0,C 180,E1 -31603.638,E2 -31603.638} C_VEL
LIN {X 0,Y 71.101,Z 466.31,A -85,B 0,C 180,E1 -31591.544,E2 -31591.544} C_VEL
LIN {X 0,Y 73.206,Z 466.252,A -85,B 0,C 180,E1 -31590,E2 -31590} C_VEL
LIN {X 0,Y 63.39,Z 466.175,A -85,B 0,C 180,E1 -31581.323,E2 -31581.323} C_VEL
LIN {X 0,Y 61.495,Z 466.18,A -85,B 0,C 180,E1 -31580.388,E2 -31580.388} C_VEL
LIN {X 0,Y 58.23,Z 466.344,A -85,B 0,C 180,E1 -31580.669,E2 -31580.669} C_VEL
LIN {X 0,Y 54.618,Z 466.628,A -85,B 0,C 180,E1 -31582.725,E2 -31582.725} C_VEL
LIN {X 0,Y 52.38,Z 466.821,A -85,B 0,C 180,E1 -31585.285,E2 -31585.285} C_VEL
LIN {X 0,Y 51.218,Z 466.822,A -85,B 0,C 180,E1 -31588.595,E2 -31588.595} C_VEL
LIN {X 0,Y 52.181,Z 466.683,A -85,B 0,C 180,E1 -31597.74,E2 -31597.74} C_VEL
LIN {X 0,Y 54.083,Z 466.505,A -85,B 0,C 180,E1 -31599.18,E2 -31599.18} C_VEL
LIN {X 0,Y 62.625,Z 466.539,A -85,B 0,C 180,E1 -31590,E2 -31590} C_VEL
LIN {X 0,Y 54.097,Z 466.505,A -85,B 0,C 180,E1 -31580.837,E2 -31580.837} C_VEL
LIN {X 0,Y 52.212,Z 466.682,A -85,B 0,C 180,E1 -31582.264,E2 -31582.264} C_VEL
LIN {X 0,Y 51.218,Z 466.822,A -85,B 0,C 180,E1 -31588.595,E2 -31588.595} C_VEL
LIN {X 0,Y 51.027,Z 468.821,A -85,B 0,C 180,E1 -31590.772,E2 -31590.772} C_VEL
LIN {X 0,Y 51.027,Z 600,A -85,B 0,C 180,E1 -31590.772,E2 -31590.772} C_VEL
LIN {X 0,Y 51.027,Z 600,A -85,B 0,C 180,E1 -31590.772,E2 -31590.772}

QRS_NEXT_CUT()

QRS_NEXT()
QRS_HOME()

END
